Staubli VAL3: StopLimits.pgx

program StopLimits()
begin
//*******************************************************************************
//*   ______
//*  / _____) /|
//* | |      / /
//* | | /\  / /
//* | | \ \/ /  _      Copyright (c) KEOLABS, 2016
//* | |  \__/  | |        http://www.keolabs.com
//* | |________| |
//*  \__________/
//*
//********************************************************************************
//*@file          : StopLimits
//*@author        : Yves Ragot
//*@version       : $Id: StopLimits.pgx 1648 2017-01-24 08:43:21Z yves $
//*@brief         : Stop movements if out of limits (called by CheckLimits)
//*
//*******************************************************************************/

  // stop movement
  call AsynchStop()

  //set error code
  GeneralStatus = 104
  LastErrorCode = 0

end
